PROGRAM FBD_TUTTILINJASTO
VAR
	fbRUN: RUN;
	START_TO_SORT1: FB_CONVEYOR1;
	fbSORT1: FB_TURNTABLE;
	SORT_TO_PICKNPLACE: FB_CONVEYOR1;
	fbPICKNPLACE_1: FB_PICKNPLACE;
	fbSortByWeight: FB_WEIGHT;
	WEIGHT_TO_CNC: FB_CONVEYOR1;
	WEIGHT_TO_LIQUIDS: FB_CONVEYOR1;
	
	fbSpecial1: FB_SPECIAL;
	fbSpecial2: FB_SPECIAL_2;
	SORT_TO_CNC: FB_CONVEYOR1;
	fbWheelSort1: FB_WHEELSORT;
	fbCNCMill1: FB_CNC_MILL;
	fbCNCMill2: FB_CNC_MILL;
	fbCNCMill3: FB_CNC_MILL;
	CNC_TO_BOXING: FB_CONVEYOR1;
	BOXING_TO_STORAGE: FB_CONVEYOR1;
	fbClamp: FB_CLAMP;
	fbTwoAxisPick1: FB_TWO_AXIS_PICK;
	fbStacker1: FB_STACKER;
END_VAR

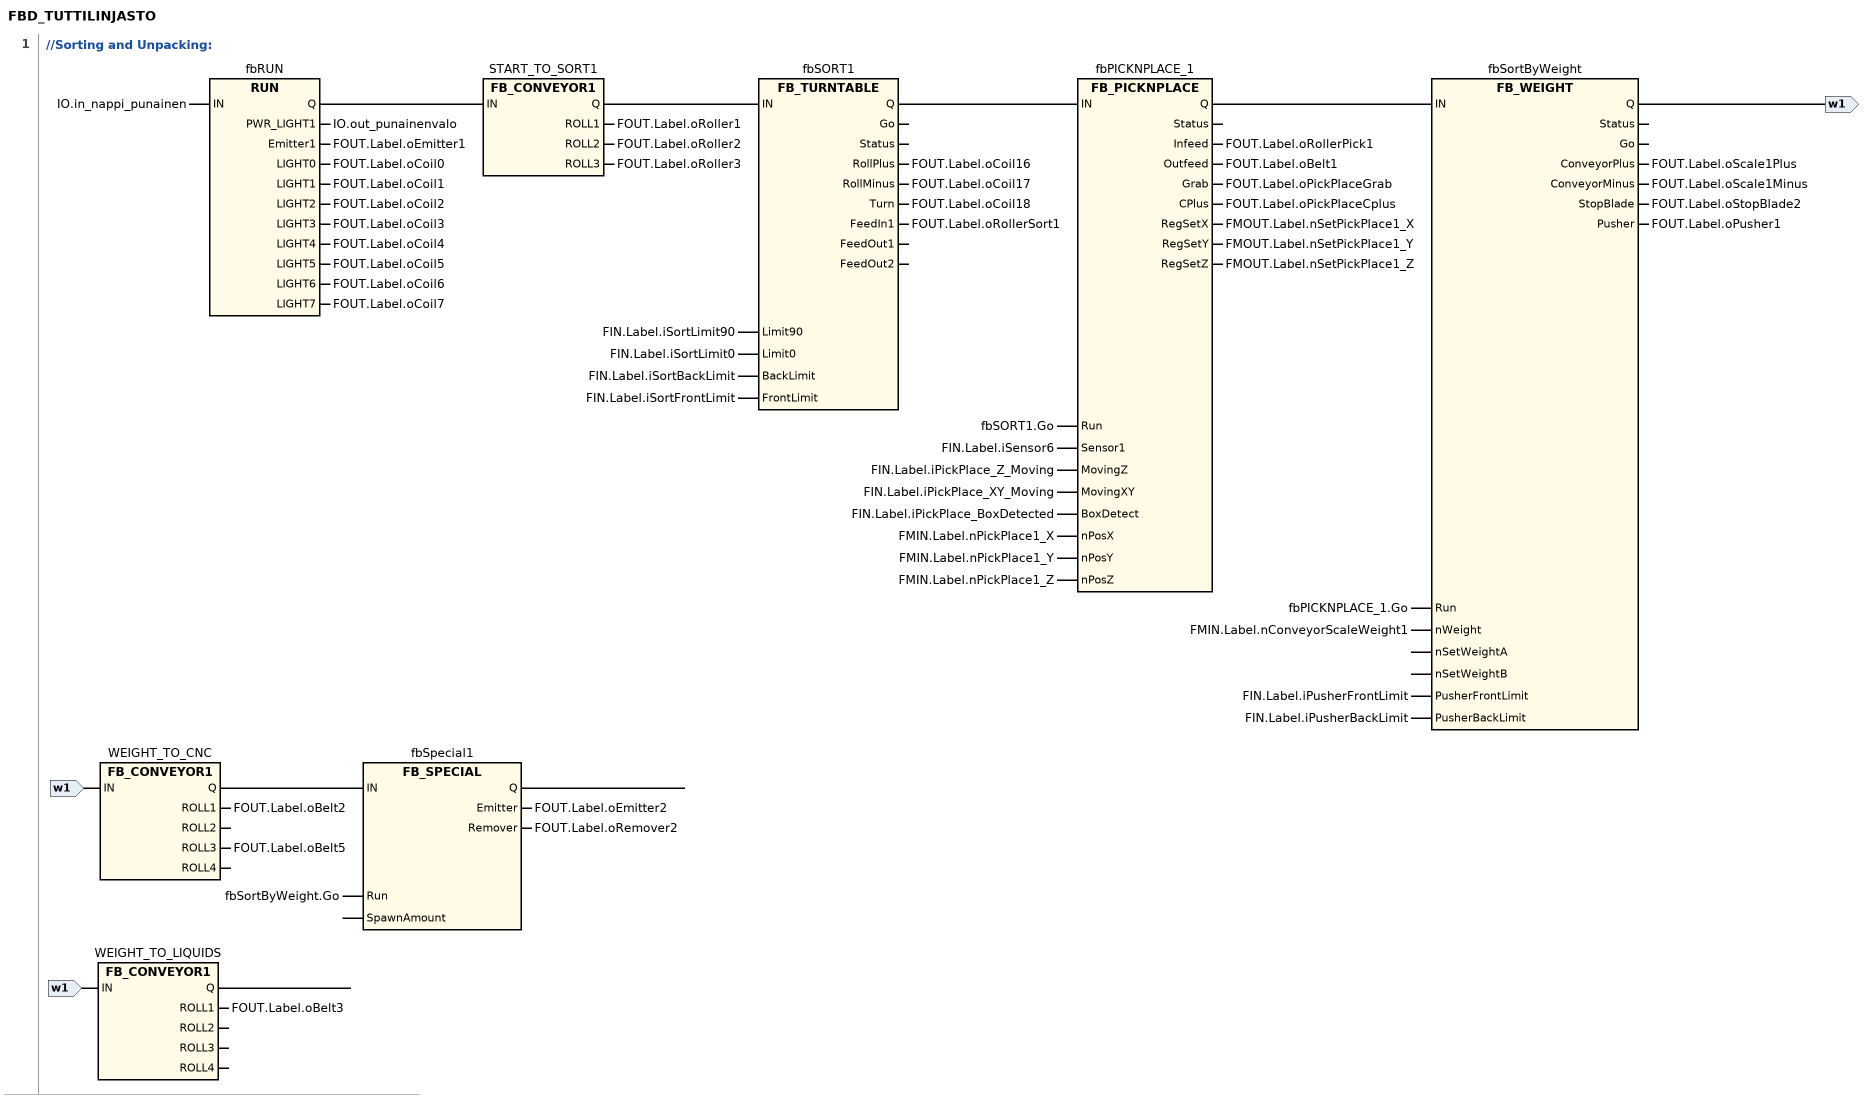
// NETWORK 1
// label: //Sorting and Unpacking
fbRUN(
    IN := IO.in_nappi_punainen,
    PWR_LIGHT1 => IO.out_punainenvalo,
    Emitter1 => FOUT.Label.oEmitter1,
    LIGHT0 => FOUT.Label.oCoil0,
    LIGHT1 => FOUT.Label.oCoil1,
    LIGHT2 => FOUT.Label.oCoil2,
    LIGHT3 => FOUT.Label.oCoil3,
    LIGHT4 => FOUT.Label.oCoil4,
    LIGHT5 => FOUT.Label.oCoil5,
    LIGHT6 => FOUT.Label.oCoil6,
    LIGHT7 => FOUT.Label.oCoil7); // RUN
START_TO_SORT1(
    IN := fbRUN.Q,
    ROLL1 => FOUT.Label.oRoller1,
    ROLL2 => FOUT.Label.oRoller2,
    ROLL3 => FOUT.Label.oRoller3); // FB_CONVEYOR1
fbSORT1(
    IN := START_TO_SORT1.Q,
    Limit90 := FIN.Label.iSortLimit90,
    Limit0 := FIN.Label.iSortLimit0,
    BackLimit := FIN.Label.iSortBackLimit,
    FrontLimit := FIN.Label.iSortFrontLimit,
    RollPlus => FOUT.Label.oCoil16,
    RollMinus => FOUT.Label.oCoil17,
    Turn => FOUT.Label.oCoil18,
    FeedIn1 => FOUT.Label.oRollerSort1); // FB_TURNTABLE
fbPICKNPLACE_1(
    IN := fbSORT1.Q,
    Run := fbSORT1.Go,
    Sensor1 := FIN.Label.iSensor6,
    MovingZ := FIN.Label.iPickPlace_Z_Moving,
    MovingXY := FIN.Label.iPickPlace_XY_Moving,
    BoxDetect := FIN.Label.iPickPlace_BoxDetected,
    nPosX := FMIN.Label.nPickPlace1_X,
    nPosY := FMIN.Label.nPickPlace1_Y,
    nPosZ := FMIN.Label.nPickPlace1_Z,
    Infeed => FOUT.Label.oRollerPick1,
    Outfeed => FOUT.Label.oBelt1,
    Grab => FOUT.Label.oPickPlaceGrab,
    CPlus => FOUT.Label.oPickPlaceCplus,
    RegSetX => FMOUT.Label.nSetPickPlace1_X,
    RegSetY => FMOUT.Label.nSetPickPlace1_Y,
    RegSetZ => FMOUT.Label.nSetPickPlace1_Z); // FB_PICKNPLACE
fbSortByWeight(
    IN := fbPICKNPLACE_1.Q,
    Run := fbPICKNPLACE_1.Go,
    nWeight := FMIN.Label.nConveyorScaleWeight1,
    PusherFrontLimit := FIN.Label.iPusherFrontLimit,
    PusherBackLimit := FIN.Label.iPusherBackLimit,
    ConveyorPlus => FOUT.Label.oScale1Plus,
    ConveyorMinus => FOUT.Label.oScale1Minus,
    StopBlade => FOUT.Label.oStopBlade2,
    Pusher => FOUT.Label.oPusher1); // FB_WEIGHT
WEIGHT_TO_CNC(IN := fbSortByWeight.Q, ROLL1 => FOUT.Label.oBelt2, ROLL3 => FOUT.Label.oBelt5); // FB_CONVEYOR1
fbSpecial1(
    IN := WEIGHT_TO_CNC.Q,
    Run := fbSortByWeight.Go,
    Emitter => FOUT.Label.oEmitter2,
    Remover => FOUT.Label.oRemover2); // FB_SPECIAL
WEIGHT_TO_LIQUIDS(IN := fbSortByWeight.Q, ROLL1 => FOUT.Label.oBelt3); // FB_CONVEYOR1

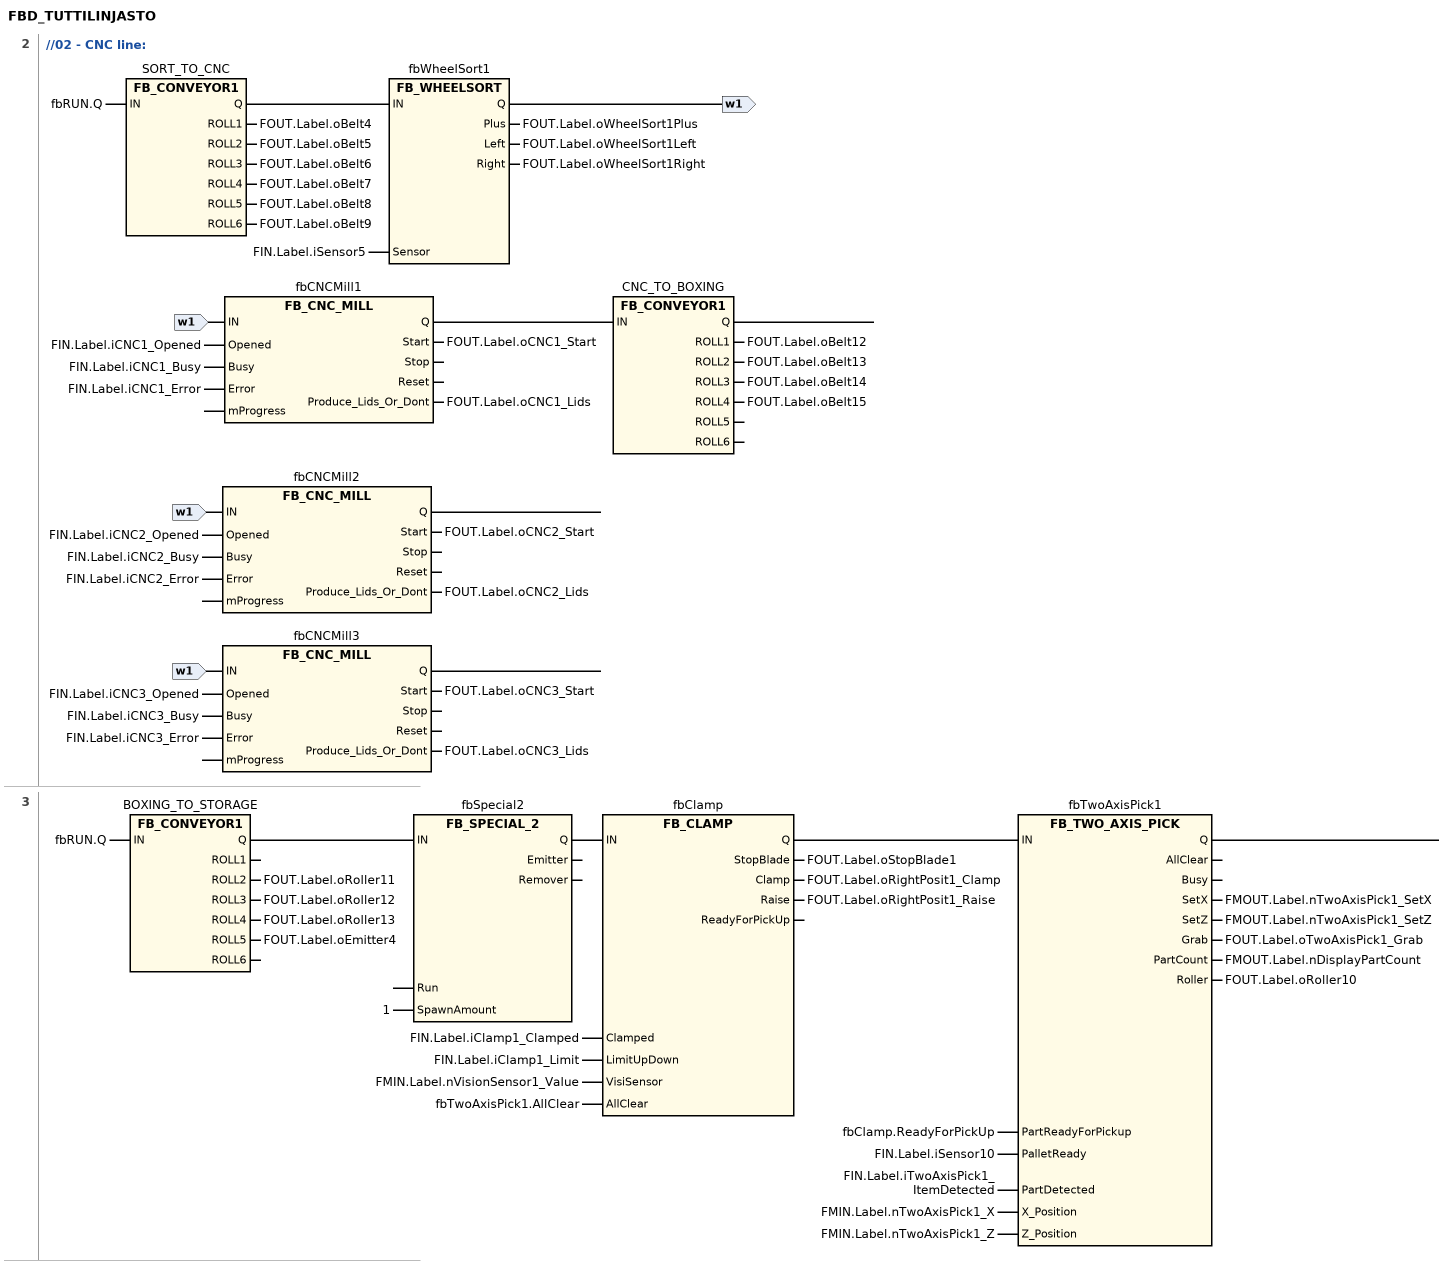
// NETWORK 2
// label: //02 - CNC line
SORT_TO_CNC(
    IN := fbRUN.Q,
    ROLL1 => FOUT.Label.oBelt4,
    ROLL2 => FOUT.Label.oBelt5,
    ROLL3 => FOUT.Label.oBelt6,
    ROLL4 => FOUT.Label.oBelt7,
    ROLL5 => FOUT.Label.oBelt8,
    ROLL6 => FOUT.Label.oBelt9); // FB_CONVEYOR1
fbWheelSort1(
    IN := SORT_TO_CNC.Q,
    Sensor := FIN.Label.iSensor5,
    Plus => FOUT.Label.oWheelSort1Plus,
    Left => FOUT.Label.oWheelSort1Left,
    Right => FOUT.Label.oWheelSort1Right); // FB_WHEELSORT
fbCNCMill1(
    IN := fbWheelSort1.Q,
    Opened := FIN.Label.iCNC1_Opened,
    Busy := FIN.Label.iCNC1_Busy,
    Error := FIN.Label.iCNC1_Error,
    Start => FOUT.Label.oCNC1_Start,
    Produce_Lids_Or_Dont => FOUT.Label.oCNC1_Lids); // FB_CNC_MILL
CNC_TO_BOXING(
    IN := fbCNCMill1.Q,
    ROLL1 => FOUT.Label.oBelt12,
    ROLL2 => FOUT.Label.oBelt13,
    ROLL3 => FOUT.Label.oBelt14,
    ROLL4 => FOUT.Label.oBelt15); // FB_CONVEYOR1
fbCNCMill2(
    IN := fbWheelSort1.Q,
    Opened := FIN.Label.iCNC2_Opened,
    Busy := FIN.Label.iCNC2_Busy,
    Error := FIN.Label.iCNC2_Error,
    Start => FOUT.Label.oCNC2_Start,
    Produce_Lids_Or_Dont => FOUT.Label.oCNC2_Lids); // FB_CNC_MILL
fbCNCMill3(
    IN := fbWheelSort1.Q,
    Opened := FIN.Label.iCNC3_Opened,
    Busy := FIN.Label.iCNC3_Busy,
    Error := FIN.Label.iCNC3_Error,
    Start => FOUT.Label.oCNC3_Start,
    Produce_Lids_Or_Dont => FOUT.Label.oCNC3_Lids); // FB_CNC_MILL

// NETWORK 3
BOXING_TO_STORAGE(
    IN := fbRUN.Q,
    ROLL2 => FOUT.Label.oRoller11,
    ROLL3 => FOUT.Label.oRoller12,
    ROLL4 => FOUT.Label.oRoller13,
    ROLL5 => FOUT.Label.oEmitter4); // FB_CONVEYOR1
fbSpecial2(IN := BOXING_TO_STORAGE.Q, SpawnAmount := 1); // FB_SPECIAL_2
fbClamp(
    IN := fbSpecial2.Q,
    Clamped := FIN.Label.iClamp1_Clamped,
    LimitUpDown := FIN.Label.iClamp1_Limit,
    VisiSensor := FMIN.Label.nVisionSensor1_Value,
    AllClear := fbTwoAxisPick1.AllClear,
    StopBlade => FOUT.Label.oStopBlade1,
    Clamp => FOUT.Label.oRightPosit1_Clamp,
    Raise => FOUT.Label.oRightPosit1_Raise); // FB_CLAMP
fbTwoAxisPick1(
    IN := fbClamp.Q,
    PartReadyForPickup := fbClamp.ReadyForPickUp,
    PalletReady := FIN.Label.iSensor10,
    PartDetected := FIN.Label.iTwoAxisPick1_ItemDetected,
    X_Position := FMIN.Label.nTwoAxisPick1_X,
    Z_Position := FMIN.Label.nTwoAxisPick1_Z,
    SetX => FMOUT.Label.nTwoAxisPick1_SetX,
    SetZ => FMOUT.Label.nTwoAxisPick1_SetZ,
    Grab => FOUT.Label.oTwoAxisPick1_Grab,
    PartCount => FMOUT.Label.nDisplayPartCount,
    Roller => FOUT.Label.oRoller10); // FB_TWO_AXIS_PICK

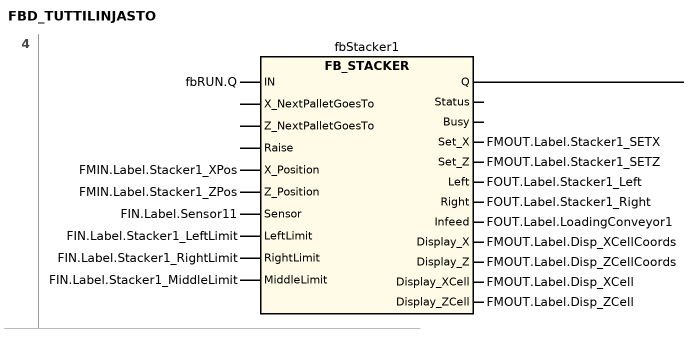
// NETWORK 4
fbStacker1(
    IN := fbRUN.Q,
    X_Position := FMIN.Label.Stacker1_XPos,
    Z_Position := FMIN.Label.Stacker1_ZPos,
    Sensor := FIN.Label.Sensor11,
    LeftLimit := FIN.Label.Stacker1_LeftLimit,
    RightLimit := FIN.Label.Stacker1_RightLimit,
    MiddleLimit := FIN.Label.Stacker1_MiddleLimit,
    Set_X => FMOUT.Label.Stacker1_SETX,
    Set_Z => FMOUT.Label.Stacker1_SETZ,
    Left => FOUT.Label.Stacker1_Left,
    Right => FOUT.Label.Stacker1_Right,
    Infeed => FOUT.Label.LoadingConveyor1,
    Display_X => FMOUT.Label.Disp_XCellCoords,
    Display_Z => FMOUT.Label.Disp_ZCellCoords,
    Display_XCell => FMOUT.Label.Disp_XCell,
    Display_ZCell => FMOUT.Label.Disp_ZCell); // FB_STACKER

END_PROGRAM

(* stored: Version 1.1.0.1, ProductVersion 3.1.4024.6
   POU FBD_TUTTILINJASTO: Id {a0bd0942-3c6b-466f-88c4-c4a92ae9071d}, SpecialFunc None *)
